PROGRAM Anlage
VAR
	Kom_Reaktor_1		:FB_Kommunikation;
	
END_VAR

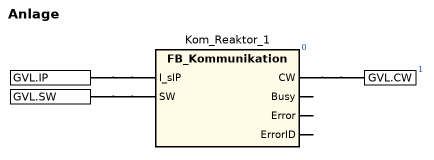
Kom_Reaktor_1(I_sIP := GVL.IP, SW := GVL.SW); // FB_Kommunikation
GVL.CW := Kom_Reaktor_1.CW;

END_PROGRAM

(* stored: Version 1.1.0.1, ProductVersion 3.1.4024.12
   POU Anlage: Id {76b1dd52-fe4d-430a-95d4-af12f5b6cd4b}, SpecialFunc None *)
